TYPE ST_Navitrol_HMI EXTENDS ST_HmiFunction :
	STRUCT
		CommunicationActive : BOOL;
		Status				: E_3102_State;
		ControlFromNavitrol : BOOL;
	END_STRUCT
END_TYPE

(* stored: Version 1.1.0.1
   DUT ST_Navitrol_HMI: Id {ade0003f-7ec7-4165-bd78-ad1212e1e5ec} *)
